ABB RAPID module: SURGERYDATA.mod

MODULE SURGERYDATA
    PERS NUM Surg_ACActive := 0;   ! Whether or not AC is active
    PERS NUM Surg_NACActive := 0;  ! Whether or not NAC is active

    !PERS clock glclock;
    PERS NUM Surg_time := 0;

    PERS robtarget Surg_StartPos := [[687.97,-810.05,304.52],[0.43869,0.800006,0.407982,0.0330496],[-1,-1,1,0],[9E+09,9E+09,9E+09,9E+09,9E+09,9E+09]];
    PERS robtarget Surg_TopPos := [[-56.4,-958.8,156.69],[0.691416,0.718403,0.0648077,-0.0404983],[-2,-1,0,1],[9E+09,9E+09,9E+09,9E+09,9E+09,9E+09]];
    PERS tooldata Surg_Tool := [TRUE,[[0,0,497],[1,0,0,0]],[0.6,[0,0,100],[1,0,0,0],0,0,0]];
    PERS loaddata Surg_Load := [0.967619, [0.104787,0.3113, 63.6271], [1, 0, 0, 0], 0, 0, 0];

    ! Special tool definitions
    PERS tooldata Surg_Poke_Tool := [TRUE,[[-1.86435,-1.96008,150.019],[1,0,0,0]],[5.5,[-1,1,1],[1,0,0,0],0,0,0]];
    PERS loaddata Surg_Poke_Load := [1.28062, [-1.57092,2.15947, 63.2874], [1, 0, 0, 0], 0, 0, 0];
    PERS robtarget Surg_Poke_StartPos := [[15.67,470.41,231.34],[0.00285824,-0.999987,-0.00107065,0.00429505],[0,0,0,0],[9E+09,9E+09,9E+09,9E+09,9E+09,9E+09]];
    PERS robtarget Surg_Poke_TopPos := [[519.67,-336.37,537.49],[0.00113577,-0.00527189,-0.913055,0.407803],[-1,0,-1,0],[9E+09,9E+09,9E+09,9E+09,9E+09,9E+09]];
    PERS loaddata Surg_Grip_Load := [0.977065,[2.8381,-1.07347,63.0716],[1,0,0,0],0,0,0];
    PERS robtarget Surg_Grip_StartPos := [[636.07,91.01,645.44],[0.508058,-0.494919,0.499625,-0.497301],[0,0,-2,1],[9E+09,9E+09,9E+09,9E+09,9E+09,9E+09]];
    PERS robtarget Surg_Grip_TopPos := [[-7.81,-794.00,184.49],[0.462462,0.555409,0.541705,-0.429192],[-2,-1,0,1],[9E+09,9E+09,9E+09,9E+09,9E+09,9E+09]];

    ! Accommodation control variables
    PERS fcdamping Surg_ACDamping := [200.0, 200.0, 250.0, 200.0, 200.0, 250.0];

	CONST speeddata vCal10 := [10,2,20,10];


	CONST robtarget Surg_TopPos10:=[[536.79,125.65,487.36],[0.0931804,0.0223058,0.995253,0.017085],[0,-1,0,0],[9E+09,9E+09,9E+09,9E+09,9E+09,9E+09]];
    PERS tooldata Surg_Grip_Tool := [TRUE,[[-0.0141472,0.0811151,217.672],[1,0,0,0]],[0.9709,[0.08759,0.317389,63.5646],[1,0,0,0],0,0,0]];
    CONST robtarget Gel_gp1 := [[614.69,-24.81,447.15],[0.702002,-0.000794548,0.712174,-0.00118308],[-1,-1,0,1],[9E+09,9E+09,9E+09,9E+09,9E+09,9E+09]];
    CONST robtarget Gel_gp2 := [[643.27,63.24,475.65],[0.600899,0.262789,0.731576,-0.186173],[0,0,-1,1],[9E+09,9E+09,9E+09,9E+09,9E+09,9E+09]];
    CONST robtarget Gel_gp3 := [[645.14,-112.04,442.60],[0.690012,-0.259974,0.650756,0.181147],[-1,-1,0,1],[9E+09,9E+09,9E+09,9E+09,9E+09,9E+09]];
    CONST robtarget Gel_gp4 := [[755.55,119.15,442.98],[0.47342,0.463746,0.52551,-0.53353],[0,1,-1,1],[9E+09,9E+09,9E+09,9E+09,9E+09,9E+09]];
    CONST robtarget Gel_gp5 := [[638.60,50.87,498.16],[0.572423,0.390266,0.721121,0.00313459],[0,1,-1,1],[9E+09,9E+09,9E+09,9E+09,9E+09,9E+09]];
    CONST robtarget Gel_gp6 := [[661.63,60.25,532.97],[0.453746,0.432061,0.776017,-0.0723608],[0,1,-1,1],[9E+09,9E+09,9E+09,9E+09,9E+09,9E+09]];
    CONST robtarget Gel_gp7 := [[614.08,-30.60,453.38],[0.648948,0.173276,0.698732,0.246203],[-1,-1,0,1],[9E+09,9E+09,9E+09,9E+09,9E+09,9E+09]];
    CONST robtarget Gel_gp8 := [[615.77,-45.76,450.78],[0.693561,-0.11317,0.710957,-0.0265877],[-1,-1,0,1],[9E+09,9E+09,9E+09,9E+09,9E+09,9E+09]];
    CONST robtarget Gel_gp9 := [[615.27,-44.81,476.13],[0.626024,-0.0494511,0.776689,0.0490308],[-1,-1,0,1],[9E+09,9E+09,9E+09,9E+09,9E+09,9E+09]];
    CONST robtarget pasu := [[615.67,87.62,299.21],[0.70710678,0,0.70710678,0],[0,0,-1,1],[9E+09,9E+09,9E+09,9E+09,9E+09,9E+09]];
    PERS tooldata Surg_Grip_Green := [TRUE,[[-20.4343,0.52221,143.947],[1,0,0,0]],[0.9709,[0.08759,0.317389,63.5646],[1,0,0,0],0,0,0]];
    PERS tooldata Surg_Grip_Marker := [TRUE,[[-20.4343,0.52221,143.947],[1,0,0,0]],[0.9709,[0.08759,0.317389,63.5646],[1,0,0,0],0,0,0]];
    PERS tooldata Surg_Grip_Mark2 := [TRUE,[[-20.4343,0.52221,143.947],[1,0,0,0]],[0.9709,[0.08759,0.317389,63.5646],[1,0,0,0],0,0,0]];
    PERS tooldata Surg_Grip_Marker_1 := [TRUE,[[-0.0141472,0.0811151,217.672],[1,0,0,0]],[0.9709,[0.08759,0.317389,63.5646],[1,0,0,0],0,0,0]];
    PERS tooldata Surg0 := [TRUE,[[0,0,0],[1,0,0,0]],[0.001,[1E-05,0,0],[1,0,0,0],0,0,0]];
    PERS errstr errstr1 := "Death notice";
    PERS loaddata Surg0_Load := [0.967619,[0.104787,0.3113,63.6271],[1,0,0,0],0,0,0];
    PERS robtarget Surg_Wrist_TopPos:=[[0.00,-579.56,277.46],[0.706421,0.706445,0.0308595,-0.0308599],[-2,-1,0,1],[9E+09,9E+09,9E+09,9E+09,9E+09,9E+09]];
    CONST zonedata zone01:=[FALSE,1,1,1,1,1,1];
	CONST zonedata zone02:=[FALSE,2,2,2,2,2,2];
	CONST zonedata zone03:=[FALSE,3,3,3,3,3,3];
	CONST zonedata zone04:=[FALSE,4,4,4,4,4,4];
	CONST zonedata zone05:=[FALSE,5,5,5,5,5,5];

    ! Natural admittance control variables
    !PERS nacvirdamping Surg_NACDamping := [400, 400, 100, 100, 100, 100];
    !PERS nacvirstiffness Surg_NACStiffness := [200, 200, 200, 300, 300, 300];
    !PERS nactarginertia Surg_NACInertia := [2, 2, 30, 15, 15, 15];
    !PERS num Surg_NACVelGainRatio := 0.1;
    !CONST robtarget Surg_Cal_Pose := [[-33.49,-600.86,307.88],[0.389574,-0.203642,-0.889693,0.123327],[-2,-1,-1,0],[9E+09,9E+09,9E+09,9E+09,9E+09,9E+09]];
    !CONST speeddata vCal10 := [10,2,20,10];
    !PERS tooldata Grip_temp := [TRUE,[[-19.4343,28.3162,136.897],[0.263453,-0.00494036,0.00769184,-0.964629]],[1,[0,0,0],[1,0,0,0],0,0,0]];
    !CONST robtarget ctes := [[737.08,93.11,205.84],[0.345425,-0.564976,0.683331,0.307477],[0,0,-1,1],[9E+09,9E+09,9E+09,9E+09,9E+09,9E+09]];
    !PERS tooldata Surg_grip_bak := [TRUE,[[-2.73067,-10.2923,155.947],[0.787942,-0.587304,-0.148321,0.110553]],[1.1,[28.7,0,151.8],[1,0,0,0],0,0.002,0.026]];
    !PERS tooldata Surg_Grip_Tool_1 := [TRUE,[[-6.72232,-15.5488,150.237],[1,0,0,0]],[-1,[0,0,0],[1,0,0,0],0,0,0]];
ENDMODULE
